(* CODESYS project _03_NVL_sender.xml

Project tree, tasks and I/O mapping:
  global variables _03_NVL_sender
*)

// _03_NVL_sender
{attribute 'qualified_only'}
VAR_GLOBAL
	someInteger : INT; //Integer value
END_VAR
